Staubli VAL3: PointGrey.dtx

public bool bCalibrating
bool bDebug
public bool bTaskDetOK = true
num hCamTable = 1
num nLatchedValue[10]
public num nMaxNumOfObject = 10
public num nNumOfPart = -1
num nObjectID[10]
  [0] = 1
  [1] = -1
  [2] = -1
  [3] = -1
  [4] = -1
  [5] = -1
  [6] = -1
  [7] = -1
  [8] = -1
  [9] = -1
object oTempQueue[10]
  [0]
    num nID = 1
    num nLatchedValue
    trsf trTrsf = {x=10, y=9, rz=97.2}
  [1]
    num nID = 1
    num nLatchedValue
    trsf trTrsf = {x=-195, y=116, rz=12.6}
  [2]
    num nID = 1
    num nLatchedValue
    trsf trTrsf = {x=-78, y=-10, rz=114.9}
  [3]
    num nID = 1
    num nLatchedValue
    trsf trTrsf = {x=-136, y=40, rz=85.3}
  [4]
    num nID = 1
    num nLatchedValue
    trsf trTrsf = {x=-186, y=-47, rz=38.4}
  [5]
    num nID
    num nLatchedValue
    trsf trTrsf
  [6]
    num nID
    num nLatchedValue
    trsf trTrsf
  [7]
    num nID
    num nLatchedValue
    trsf trTrsf
  [8]
    num nID
    num nLatchedValue
    trsf trTrsf
  [9]
    num nID
    num nLatchedValue
    trsf trTrsf
screen scVision
sio skVision = {link=Socket\PointGrey}
string sDetNum = "DET0"
string sTASK = "detect0"
string strError
trsf trObjectPos[10] = {x=10, y=9, rz=97.2}
